PROGRAM randomSensors
VAR
	DRAND : DRAND;
	Seed : INT;
	Random : LREAL;
END_VAR

Seed := 57; //Set the seed for the random function to some INT
DRAND.Seed := Seed;
DRAND();
Random := DRAND.Num;


IF Random <= 0.200 THEN //Should average once in every 5 seconds (scan time = 1 second, .20/1 probability, 20%
	IF Random <= 0.025 THEN
		Glbl.northStraightSensor := TRUE;
		Glbl.northStraightSensorCnt := Glbl.northStraightSensorCnt + 1;
	ELSIF Random <= 0.050 THEN
		Glbl.northLeftSensor := TRUE;
		Glbl.northLeftSensorCnt := Glbl.northLeftSensorCnt + 1;
	ELSIF Random <= 0.075 THEN
		Glbl.southStraightSensor := TRUE;
		Glbl.southStraightSensorCnt := Glbl.southStraightSensorCnt + 1;
	ELSIF Random <= 0.100 THEN
		Glbl.southLeftSensor := TRUE;
		Glbl.southLeftSensorCnt := Glbl.southLeftSensorCnt + 1;
	ELSIF Random <= 0.125 THEN
		Glbl.eastStraightSensor := TRUE;
		Glbl.eastStraightSensorCnt := Glbl.eastStraightSensorCnt + 1;
	ELSIF Random <= 0.150 THEN
		Glbl.eastLeftSensor := TRUE;
		Glbl.eastLeftSensorCnt := Glbl.eastLeftSensorCnt + 1;
	ELSIF Random <= 0.175 THEN
		Glbl.westStraightSensor := TRUE;
		Glbl.westStraightSensorCnt := Glbl.westStraightSensorCnt + 1;
	ELSE
		Glbl.westLeftSensor := TRUE;
		Glbl.westLeftSensorCnt := Glbl.westLeftSensorCnt + 1;
	END_IF
END_IF

END_PROGRAM

(* stored: Version 1.1.0.1, ProductVersion 3.1.4022.10
   POU randomSensors: Id {a16d454e-9d16-4279-ad6c-1b2abb729478}, SpecialFunc None *)
